(*
SPDX-FileCopyrightText: © 2026 Oleksandr Tiutyk <trofimich@gmail.com>
SPDX-License-Identifier: MIT
License: https://opensource.org/license/mit
*)

(*!
<summary>Provides shared exception metadata and formatting for task-owned clones.</summary>
<description>
Registered dynamic descendants are owned by DynamicMemoryManager until cleanup; static instances remain
caller-owned. Clone overrides must register each new instance through
DynamicMemoryManager.RegisterAutoDisposedObject after __NEW and before copying fields. Plain __NEW does not
register an instance. Each dynamic exception belongs to the cyclic PLC task that created it; do not pass
exception objects between tasks. Do not throw or create dynamic exceptions during application FB_init. Static
templates remain supported. Clone implementations must return an IException-compatible object; clients borrow
registered clones. GetRootException returns a borrowed read-only view without extending its lifetime.
SourceFullPOUName and SourcePosition expose borrowed storage for reading only; callers must not modify it.
Source names formatted by GetFullPOUName are truncated to 128 characters without raising a formatting overflow
exception.
</description>
*)

{attribute 'enable_dynamic_creation'}
{attribute 'no_explicit_call' := 'do not call this function block directly'}
FUNCTION_BLOCK ABSTRACT Exception EXTENDS Object IMPLEMENTS IException
VAR
	_SourceFullPOUName : STRING(128);
	_SourcePosition : STRING(32);
	_LocalTimestamp : LDATE_AND_TIME;	
	_UtcTimestamp : LDATE_AND_TIME;	
	
END_VAR

(*!
<summary>Appends the selected timestamp description to a target string buffer.</summary>
<description>
Hidden mode leaves the target unchanged; otherwise appends the supplied local or UTC timestamp, with a UTC
suffix for UTC mode. Formats without dynamic memory allocation; target capacity is respected with fitting
truncation where applicable. Descendants cannot replace this shared metadata formatter; custom diagnostic
payload formatting belongs in GetMessage or ToError.
</description>
<param name="targetMessage">Writable target string buffer to append to.</param>
*)
METHOD PROTECTED FINAL AppendTimestampDescription
VAR_IN_OUT
	targetMessage : ERROR_MESSAGE;	
END_VAR
VAR_INPUT
	timestampDisplayMode : TIMESTAMP_DISPLAY_MODE := TIMESTAMP_DISPLAY_MODE.HIDDEN;
	localTimestamp : LDATE_AND_TIME;	
	utcTimestamp : LDATE_AND_TIME;	
END_VAR
VAR
	targetMessagePointer : POINTER TO ERROR_MESSAGE;
	
	timeStampString : WSTRING(40);
END_VAR
IF timestampDisplayMode = TIMESTAMP_DISPLAY_MODE.HIDDEN THEN
	RETURN;
END_IF

CASE timestampDisplayMode OF
	TIMESTAMP_DISPLAY_MODE.LOCAL:
		timeStampString := TO_WSTRING(localTimestamp);
	
	TIMESTAMP_DISPLAY_MODE.UTC:
		timeStampString := TO_WSTRING(utcTimestamp);
END_CASE

timeStampString := Tc2_Standard.WLEFT(STR := Tc2_Standard.WDELETE(STR := timeStampString, LEN := 4, POS := 1), SIZE := 22);

targetMessagePointer := ADR(targetMessage);

IF timestampDisplayMode = TIMESTAMP_DISPLAY_MODE.UTC THEN
	WideStrings.AppendFit255(targetMessagePointer^, timeStampString, "UTC");
ELSE
	WideStrings.AppendFit255(targetMessagePointer^, timeStampString);
END_IF
END_METHOD

(*!
<summary>Resets source and timestamps. Descendants clear their own payload and call this implementation.</summary>
<description>
Resets timestamps to LongDateAndTimes.EPOCH. Does not delete the instance or unregister it from automatic
cleanup.
</description>
*)

METHOD Clear
_SourceFullPOUName := '';
_SourcePosition := '';
_LocalTimestamp := LongDateAndTimes.EPOCH;	
_UtcTimestamp := LongDateAndTimes.EPOCH;
END_METHOD

(*!
<summary>Creates an independent task-managed exception snapshot.</summary>
<description>
Concrete descendants allocate and register the clone with DynamicMemoryManager before copying its state. The
manager owns the clone until task cleanup; callers borrow it and must not delete it. Allocation failure
follows the terminal allocation-failure policy.
</description>
*)
METHOD ABSTRACT Clone : IObject
END_METHOD

(*!
<summary>Reports whether the concrete exception contains an error.</summary>
<description>
Concrete descendants define which stored fields make an exception nonempty. Reading does not clear or modify
it.
</description>
*)
{attribute 'monitoring' := 'call'}
PROPERTY ABSTRACT Empty : BOOL
GET
END_GET
END_PROPERTY

(*!
<summary>Extracts the first component yielded by splitting a POU name on dots.</summary>
<description>
Returns a bounded independent string extracted by in-place character scanning without dynamic memory
allocation or splitters. Descendants cannot replace this shared metadata formatter; custom diagnostic payload
formatting belongs in GetMessage or ToError.
</description>
*)
METHOD PROTECTED FINAL ExtractClassName : STRING
VAR_IN_OUT CONSTANT
	sourcePOUName : STRING;
END_VAR
VAR
	i : INT;
	length : INT;
	stringPointer : POINTER TO BYTE;
END_VAR
length := TO_INT(Tc2_Standard.LEN(STR := sourcePOUName));

IF length = 0 THEN
	ExtractClassName := '';
	RETURN;
END_IF

stringPointer := ADR(sourcePOUName);

FOR i := 0 TO length - 1 DO
	IF stringPointer[i] = 16#2E THEN
		ExtractClassName := Tc2_Standard.LEFT(STR := sourcePOUName, SIZE := i);
		RETURN;
	END_IF
END_FOR

ExtractClassName := sourcePOUName;
END_METHOD

(*!
<summary>Extracts the last component yielded by splitting a POU name on dots.</summary>
<description>
Returns a bounded independent string extracted by in-place character scanning without dynamic memory
allocation or splitters. Descendants cannot replace this shared metadata formatter; custom diagnostic payload
formatting belongs in GetMessage or ToError.
</description>
*)
METHOD PROTECTED FINAL ExtractMethodName : STRING
VAR_IN_OUT CONSTANT
	sourcePOUName : STRING;
END_VAR
VAR
	i : INT;
	length : INT;
	strngPointer : POINTER TO BYTE;
END_VAR
length := TO_INT(Tc2_Standard.LEN(STR := sourcePOUName));

IF length = 0 THEN
	ExtractMethodName := '';
	RETURN;
END_IF

strngPointer := ADR(sourcePOUName);

FOR i := length - 1 TO 0 BY -1 DO
	IF strngPointer[i] = 16#2E THEN
		ExtractMethodName := Tc2_Standard.RIGHT(STR := sourcePOUName, SIZE := length - 1 - i);
		RETURN;
	END_IF
END_FOR

ExtractMethodName := sourcePOUName;
END_METHOD

(*!
<summary>Clears exception state during destruction.</summary>
<description>
Calls Clear; descendant cleanup must not raise or create exceptions. Referenced exceptions follow their own
ownership rules and must not be deleted merely because they are referenced.
</description>
*)
//!<param name="bInCopyCode">
//! if TRUE, the exit method is called for exiting an instance that is copied afterwards (online change).
//! </param>

METHOD FB_exit : BOOL
VAR_INPUT
	
	bInCopyCode	: BOOL;
END_VAR
Clear();
END_METHOD

(*!
<summary>Formats the namespace, class and POU name for exception diagnostics.</summary>
<description>
With a class name, uses the last nonempty POU name segment as the method name and appends parentheses. Returns
the first 128 characters when the full name exceeds the result capacity; truncation does not raise an
exception. Descendants cannot replace this shared metadata formatter; custom diagnostic payload formatting
belongs in GetMessage or ToError.
</description>
*)

METHOD PROTECTED FINAL GetFullPOUName : STRING(128)
VAR_IN_OUT CONSTANT
	sourceNamespaceName : STRING;
	sourceClassName : STRING;
	sourcePOUName : STRING;
END_VAR
IF sourceNamespaceName <> Strings.Empty THEN
	GetFullPOUName := Tc2_Standard.LEFT(STR := Tc2_Standard.CONCAT(STR1 := GetFullPOUName, STR2 := sourceNamespaceName), SIZE := 128);
	GetFullPOUName := Tc2_Standard.LEFT(STR := Tc2_Standard.CONCAT(STR1 := GetFullPOUName, STR2 := '.'), SIZE := 128);
END_IF

IF sourceClassName <> Strings.Empty THEN
	GetFullPOUName := Tc2_Standard.LEFT(STR := Tc2_Standard.CONCAT(STR1 := GetFullPOUName, STR2 := sourceClassName), SIZE := 128);
	GetFullPOUName := Tc2_Standard.LEFT(STR := Tc2_Standard.CONCAT(STR1 := GetFullPOUName, STR2 := '.'), SIZE := 128);
	GetFullPOUName := Tc2_Standard.LEFT(
		STR := Tc2_Standard.CONCAT(
			STR1 := GetFullPOUName,
			STR2 := ExtractMethodName(sourcePOUName := sourcePOUName)
		),
		SIZE := 128
	);
	GetFullPOUName := Tc2_Standard.LEFT(STR := Tc2_Standard.CONCAT(STR1 := GetFullPOUName, STR2 := '()'), SIZE := 128);
ELSE
	GetFullPOUName := Tc2_Standard.LEFT(STR := Tc2_Standard.CONCAT(STR1 := GetFullPOUName, STR2 := sourcePOUName), SIZE := 128);
END_IF
END_METHOD

(*!
<summary>Formats the exception as bounded diagnostic text.</summary>
<description>
Returns an independent ERROR_MESSAGE. showSource requests available source information; timestampDisplayMode
selects a stored timestamp or hides it. Concrete exception types define their message composition; unavailable
native throw-source information cannot be reconstructed.
</description>
*)
METHOD ABSTRACT GetMessage : ERROR_MESSAGE
VAR_INPUT
	showSource : BOOL := FALSE;
	timestampDisplayMode : TIMESTAMP_DISPLAY_MODE := TIMESTAMP_DISPLAY_MODE.HIDDEN;
END_VAR
END_METHOD

(*!
<summary>Returns a borrowed read-only view of the root exception.</summary>
<description>
No clone is created and ownership is not transferred. The view does not extend the exception's lifetime and
does not expose Clear.
</description>
*)

METHOD ABSTRACT GetRootException : IReadOnlyException
END_METHOD

(*!
<summary>Formats the available exception source description.</summary>
<description>
Returns an independent bounded string without heap allocation. Native exceptions without original throw-site
information return the unspecified-source marker; catch-point information is not an original throw site.
Descendants cannot replace this shared metadata formatter; custom diagnostic payload formatting belongs in
GetMessage or ToError.
</description>
*)
METHOD FINAL GetSourceDescription : STRING(255)
IF _SourcePosition <> Strings.Empty THEN
	GetSourceDescription := Strings.Concat255(_SourceFullPOUName, TO_STRING(Exceptions.SOURCE_POSITION_PREFIX), _SourcePosition);
ELSE
	GetSourceDescription := _SourceFullPOUName;
END_IF
END_METHOD

(*!
<summary>Provides the stored local timestamp of this exception.</summary>
<description>
Framework exceptions capture it when thrown; native exceptions capture it when GetLastException obtains their
description. Cloning preserves the timestamp; reading it does not read the current clock.
</description>
*)
{attribute 'monitoring' := 'call'}
PROPERTY FINAL LocalTimestamp : LDATE_AND_TIME
GET
LocalTimestamp := _LocalTimestamp;
END_GET
SET // PROTECTED
_LocalTimestamp := LocalTimestamp;
END_SET
END_PROPERTY

(*!
<summary>Provides the source POU name for reading without copying.</summary>
<description>
The reference borrows storage from the live exception and must not outlive it. Callers must not modify the
referenced string; ST does not enforce this restriction. This is a live view, not a snapshot: changes to the
exception can change the observed value.
</description>
*)

{attribute 'monitoring' := 'call'}
PROPERTY FINAL SourceFullPOUName : REFERENCE TO STRING(128)
GET
SourceFullPOUName REF= _SourceFullPOUName;
END_GET
END_PROPERTY

(*!
<summary>Provides the source position for reading without copying.</summary>
<description>
The reference borrows storage from the live exception and must not outlive it. Callers must not modify the
referenced string; ST does not enforce this restriction. This is a live view, not a snapshot: changes to the
exception can change the observed value.
</description>
*)

{attribute 'monitoring' := 'call'}
PROPERTY FINAL SourcePosition : REFERENCE TO STRING(32)
GET
SourcePosition REF= _SourcePosition;
END_GET
END_PROPERTY

(*!
<summary>Copies exception diagnostics and timestamps into an ERROR value.</summary>
<description>
An invalid target reference is ignored. Otherwise fills both top and root descriptions from this exception
using the supplied severity and stored timestamps. Formats the source and message once each and copies the
same results into both descriptions. Formatting uses default source and timestamp display options. The target
retains copied text, not an exception reference; formatting may follow the allocation-failure policy of the
concrete formatter.
</description>
*)
METHOD ToError
VAR_IN_OUT CONSTANT
	targetError : ERROR;
END_VAR
VAR_INPUT
	severity : ERROR_SEVERITY;	
END_VAR
VAR
	topSourceText : STRING(255);
	topMessageText : ERROR_MESSAGE;
END_VAR
IF NOT __ISVALIDREF(targetError) THEN
	RETURN;
END_IF

topSourceText := GetSourceDescription();
topMessageText := GetMessage();

targetError.Fill(
	severity := severity,
	topSource := topSourceText,
	rootSource := topSourceText,
	topMessage := topMessageText,
	rootMessage := topMessageText,
	localTimestamp := LocalTimestamp,
	utcTimestamp := UtcTimestamp
);
END_METHOD

(*!
<summary>Provides the stored UTC timestamp of this exception.</summary>
<description>
Framework exceptions capture it when thrown; native exceptions capture it when GetLastException obtains their
description. Cloning preserves the timestamp; reading it does not read the current clock.
</description>
*)
{attribute 'monitoring' := 'call'}
PROPERTY FINAL UtcTimestamp : LDATE_AND_TIME
GET
UtcTimestamp := _UtcTimestamp;
END_GET
SET // PROTECTED
_UtcTimestamp := UtcTimestamp;
END_SET
END_PROPERTY

END_FUNCTION_BLOCK

(* stored: Version 1.1.0.1
   POU Exception: Id {54495eb3-7b3a-47b9-85cb-0393f41c20d3}, SpecialFunc None
   Folder Service members: Id {a47a20ca-4953-4e09-8f4d-fc2e8d3ac96e}
   Method AppendTimestampDescription: Id {a316d3b4-0094-41d5-a4cb-9fba6e2a6883}
   Method Clear: Id {44a047f7-46bd-418c-989f-4458402150ba}
   Method Clone: Id {ff7ec3e0-b6aa-4a29-8b78-e576a86138cb}
   Property Empty: Id {bd97cee3-a16c-4148-a36f-41860b6b4283}
   Get Get: Id {32775313-ab40-46b6-a69f-434f332e1416}
   Method ExtractClassName: Id {2741f852-3263-48be-9dbc-ba747f8558d6}
   Method ExtractMethodName: Id {be44e9a6-255a-48b7-a062-fbf15488833a}
   Method FB_exit: Id {11857425-e8b4-42f5-9cda-87a6242433d1}
   Method GetFullPOUName: Id {55af960f-b27f-4389-9e6d-9c37bf31a838}
   Method GetMessage: Id {6f101456-9a5d-4c21-8b11-8b9151d71824}
   Method GetRootException: Id {14eed042-28c1-47eb-a619-b182b2b0181c}
   Method GetSourceDescription: Id {d08299fd-3dd9-413a-badd-9a2833bcb01e}
   Property LocalTimestamp: Id {4c2d5866-231e-4105-a6bb-6c19851f1e45}
   Get Get: Id {4cb9fd2f-3b41-4625-9c08-af3725cdee6c}
   Set Set: Id {45619644-007a-4d10-a49a-4bb8ab2228ac}
   Property SourceFullPOUName: Id {ce5ba086-21af-4254-a988-84dec5648bcb}
   Get Get: Id {8170787e-91f8-4271-bfce-a70e9b6f9137}
   Property SourcePosition: Id {92080a7c-c630-4b10-82a8-4b95a8267619}
   Get Get: Id {da2e3d95-43f0-4ba4-a676-8010643e418a}
   Method ToError: Id {8d25c83e-d9af-49a8-90c4-2ced5ac3b9ee}
   Property UtcTimestamp: Id {6ae20a8f-f2b2-4c7c-96e2-30787aae9908}
   Get Get: Id {68e22629-e573-41bd-b400-d1cb3c398e1f}
   Set Set: Id {b2d25d91-e13d-48d8-a20e-cde8a5d29fe4} *)
